(* PLC project  *)

CONFIGURATION Empty_Module_11
END_CONFIGURATION
